FUNCTION FUN_GetTimestamp : STRING
VAR_INPUT
	stNtTime		:TIMESTRUCT;
END_VAR
VAR
	sTimestamp		:STRING;
END_VAR

// Add data
sTimeStamp := FUN_GetDate(stNtTime);

// Add time
sTimestamp := CONCAT(sTimeStamp, ' ');
sTimestamp := CONCAT(sTimeStamp, FUN_GetTime(stNtTime));

// Return time stamp
FUN_GetTimestamp := sTimestamp;

END_FUNCTION

(* stored: Version 1.1.0.1, ProductVersion 3.1.4024.12
   POU FUN_GetTimestamp: Id {c06274ce-7779-4e68-93a2-10c83eefe47d}, SpecialFunc None *)
